{attribute addProperty BoxType "EL3773-0000-0018"}
{attribute addProperty Id "I2_StatusAT %I*I2_Status_E2EFACF1162"}
{attribute addProperty CRC "1669786790"}
{attribute addProperty SizeInBites "16"}
{attribute addProperty SizeInBytes "2"}
TYPE L2_Current_Status_6386ECA6 :
STRUCT
	{attribute addProperty Name "I2_Status"}
	I2_Status AT %I* : I2_Status_E2EFACF1;
END_STRUCT
END_TYPE

(* stored: Version 1.2.0.0, ProductVersion 3.1.4024.9
   DUT L2_Current_Status_6386ECA6: Id {628049fd-05a6-4e6c-b78c-b0ae76c11dac} *)
